TYPE eSteps :
(
	Step_init := 0,
	Step_OpenFile:=10,
	Step_GetFile:=20,
	Step_Para:=30,
	Step_Close:=40,
	Step_Last:=100
);
END_TYPE

(* stored: Version 1.1.0.1, ProductVersion 3.1.4022.12
   EnumerationTextList eSteps: Id {72c650af-5235-4bdb-a5d4-c0e0d99b13bf} *)
